TYPE TcoSignalInfo :
STRUCT
	SymbolPath : STRING[255];
END_STRUCT
END_TYPE

(* stored: Version 1.1.0.1, ProductVersion 3.1.4024.9
   DUT TcoSignalInfo: Id {25268e03-6f9c-0c12-1687-c3af09c1cf34} *)
